Staubli VAL3: ISO_PDUsize.pgx

program ISO_PDUsize(num& x_nSize)
begin

  x_nSize = PDU.TPKT[2]
  x_nSize = x_nSize*256 + PDU.TPKT[3]

end
